{attribute addProperty BoxType "EK1122-0000-0018"}
{attribute addProperty Id "Beckhoff_AX8yxxsub_EK1100EK1100_179A0949162A_0061_AMP8000_0000_0103AMP8000_3F1F35B340851A_0061_AMP8000_0030_0103AMP8000_8C7527D258473"}
{attribute addProperty CRC "43770191"}
{attribute addProperty SizeInBites "1008"}
{attribute addProperty SizeInBytes "126"}
TYPE Beckhoff_AX8yxxEK1122_029BE14F EXTENDS EK1122_179A0949 :
STRUCT
	{attribute addProperty Name "Beckhoff_AX8yxxsub_EK1100"}
	Beckhoff_AX8yxxsub_EK1100 : EK1100_179A0949;
	{attribute addProperty Name "A_0061_AMP8000_0000_0103"}
	A_0061_AMP8000_0000_0103 : AMP8000_3F1F35B3;
	{attribute addProperty Name "A_0061_AMP8000_0030_0103"}
	A_0061_AMP8000_0030_0103 : AMP8000_8C7527D2;
END_STRUCT
END_TYPE

(* stored: Version 1.2.0.0, ProductVersion 3.1.4024.9
   DUT Beckhoff_AX8yxxEK1122_029BE14F: Id {51c6ee1e-673e-4d87-9ab4-89a2c7f60538} *)
